// TIA Portal V19 export
FUNCTION "Trapezoidal_PeekVelocity" : LReal   // FC35, LAD
// stored: Access Published, SetENOAutomatically false
   VAR_INPUT
      FeedSpace : LReal;
      AccDec : LReal;
   END_VAR
   VAR_TEMP
      Ramp_Space : LReal;
      Ramp_Time : LReal;
   END_VAR
   // Ret_Val : mm/min
BEGIN

REGION Network 1 (SCL): mm/min
   #Trapezoidal_PeekVelocity := SQRT(#FeedSpace * #AccDec) * 60.0;
END_REGION
END_FUNCTION
